// TIA Portal V18 export
DATA_BLOCK "Vitogate"   // DB1010
{ S7_Optimized_Access := 'FALSE' }
VERSION : 0.1
// stored: AutoNumber false, DBAccessibleFromOPCUA true, IsOnlyStoredInLoadMemory false, IsWriteProtectedInAS false
   VAR
      Alarms { S7_SetPoint := 'True'} : "UDT_Vitotronic100_Alarms";
      IOs { S7_SetPoint := 'True'} : "UDT_Vitotronic100_IOs";
      Params { S7_SetPoint := 'True'} : "UDT_Vitotronic100_Params";
      Settings { S7_SetPoint := 'True'} : "UDT_Vitotronic100_Settings";
   END_VAR
BEGIN
END_DATA_BLOCK
